(* Logix 5000 project; controller Lab7_1 5069-L306ERM rev 35.16; software revision 35.00 *)

TASK MainTask (continuous, watchdog 500 ms) : MainProgram

MODULES
   Local : 5069-L306ERM (5069 0, rev 35.16)
      IOHub : vendor 1 type 7 code 358 (Ethernet 192.168.110.5, rev 1.1, Output RPI 20 ms)
END_MODULES

PROGRAM MainProgram   (* main routine MainRoutine *)
VAR
   counter_0 : COUNTER;
   counter_2 : COUNTER;
   displayTimer : TIMER := (PRE := 5000);
   Dummy : BOOL;
   enable_1_sec : BOOL;
   enable_3_sec : BOOL;
   timer_1_sec : TIMER := (PRE := 1000);
   timer_3_sec : TIMER := (PRE := 3000);
END_VAR

ROUTINE MainRoutine   (* ladder *)
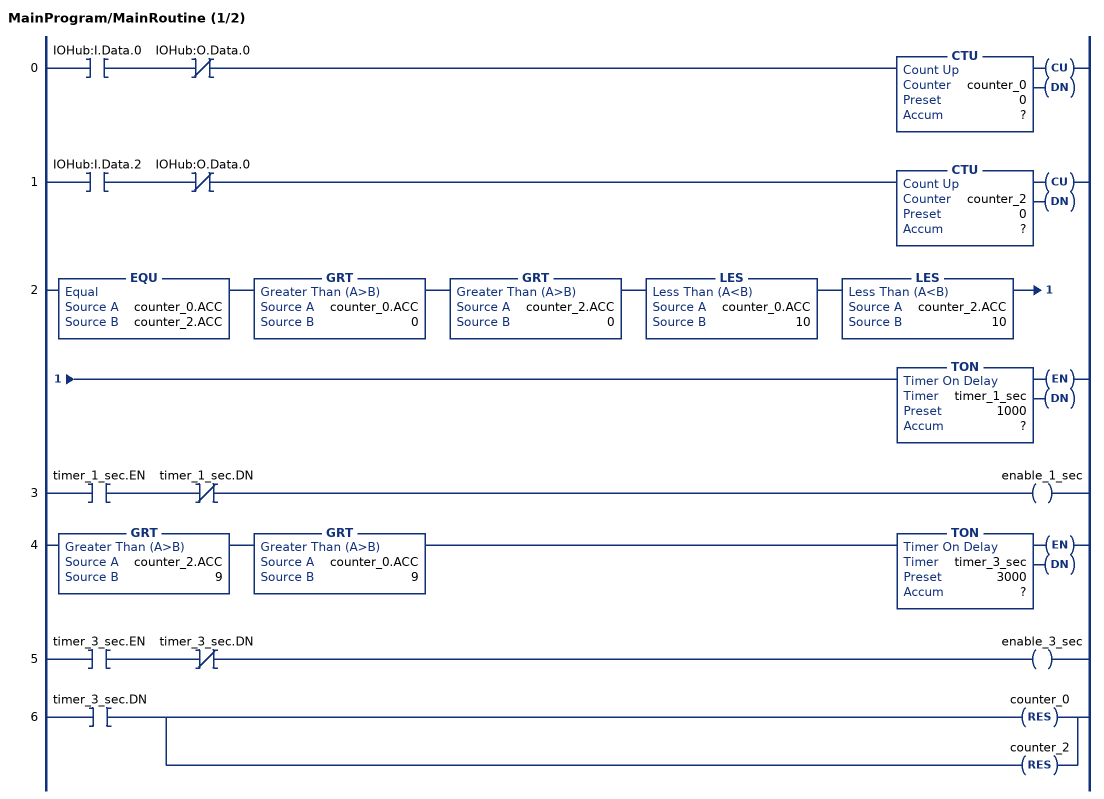
   0: XIC(IOHub:I.Data.0)XIO(IOHub:O.Data.0)CTU(counter_0,?,?);
   1: XIC(IOHub:I.Data.2)XIO(IOHub:O.Data.0)CTU(counter_2,?,?);
   2: EQU(counter_0.ACC,counter_2.ACC)GRT(counter_0.ACC,0)GRT(counter_2.ACC,0)LES(counter_0.ACC,10)LES(counter_2.ACC,10)TON(timer_1_sec,?,?);
   3: XIC(timer_1_sec.EN)XIO(timer_1_sec.DN)OTE(enable_1_sec);
   4: GRT(counter_2.ACC,9)GRT(counter_0.ACC,9)TON(timer_3_sec,?,?);
   5: XIC(timer_3_sec.EN)XIO(timer_3_sec.DN)OTE(enable_3_sec);
   6: XIC(timer_3_sec.DN)[RES(counter_0) ,RES(counter_2) ];
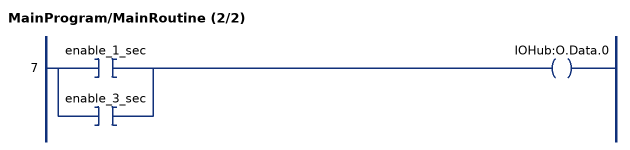
   7: [XIC(enable_1_sec) ,XIC(enable_3_sec) ]OTE(IOHub:O.Data.0);
END_ROUTINE
END_PROGRAM
